% RSLogix 500 project slc_adjust_clock.RSS, saved by version 8.30.00.16 %
PROJECT "UNTITLED"    % processor: Bul.1763 MicroLogix 1100 Series B %

PROGRAM FILES
  LAD 2   4 rungs

DATA FILES
  O0 OUTPUT  4 elements
  I1 INPUT  6 elements
  S2 STATUS  66 elements
  B3 BINARY  1 elements
  T4 TIMER  1 elements
  C5 COUNTER  1 elements
  R6 CONTROL  1 elements
  N7 INTEGER  1 elements
  F8 FLOAT  1 elements
  N101 RTCBUFFERS  18 elements

LADDER 2
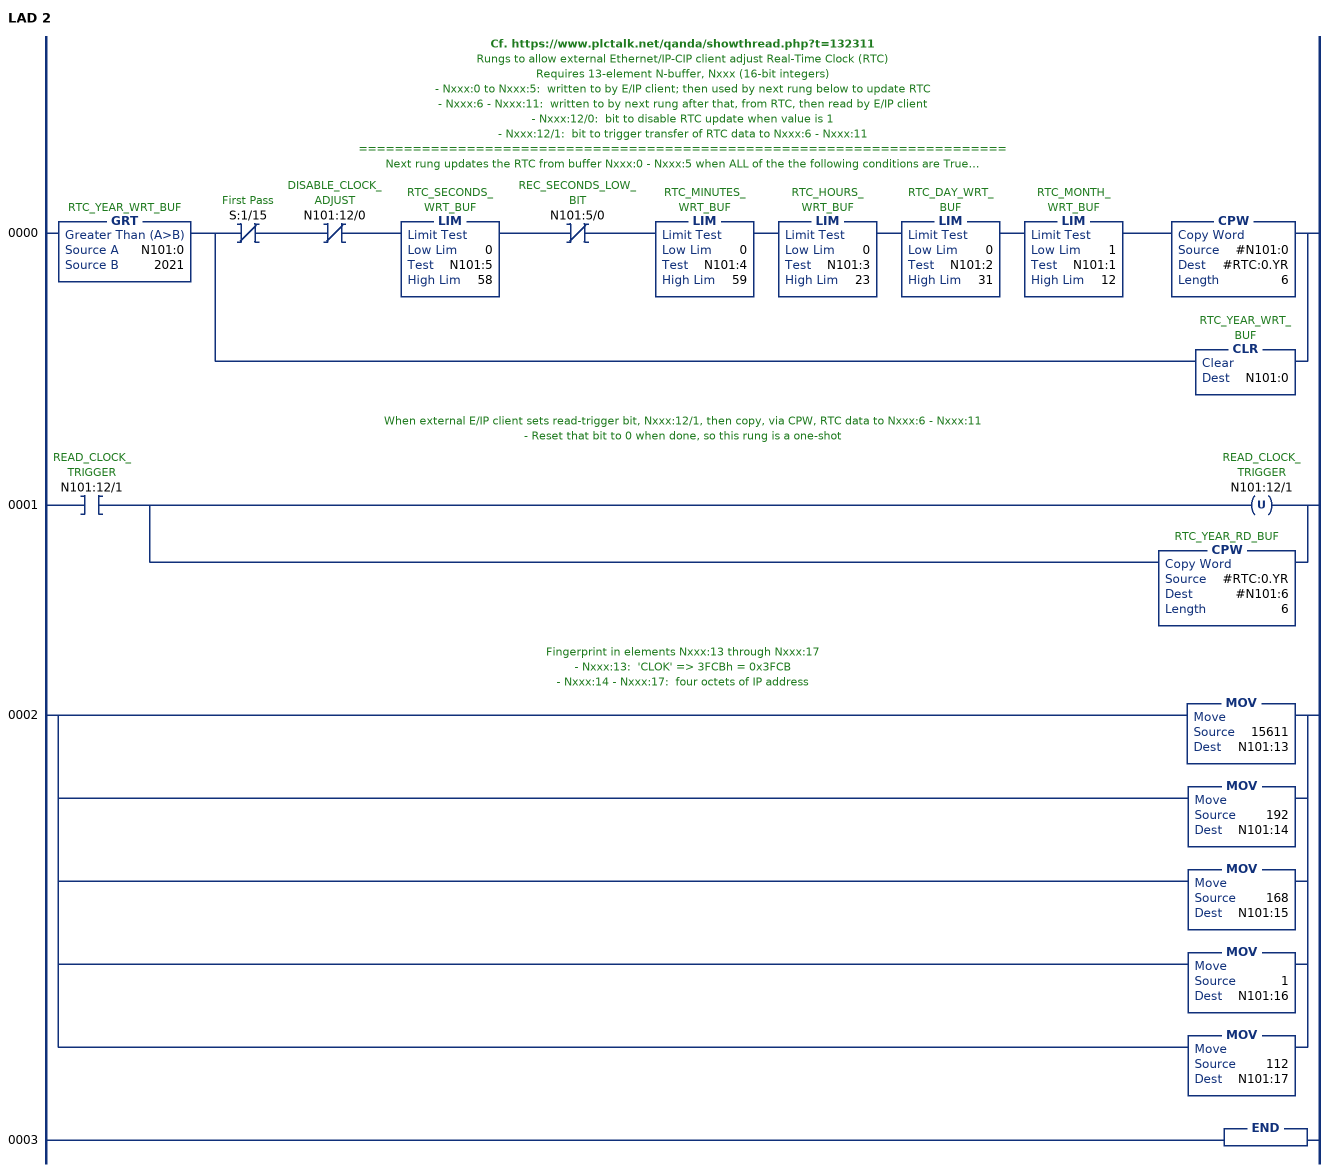
% Rung: 0 %
% TITLE: Cf. https://www.plctalk.net/qanda/showthread.php?t=132311 %
% Rungs to allow external Ethernet/IP-CIP client adjust Real-Time Clock (RTC)
% 
% Requires 13-element N-buffer, Nxxx (16-bit integers)
% - Nxxx:0 to Nxxx:5:  written to by E/IP client; then used by next rung below to update RTC
% - Nxxx:6 - Nxxx:11:  written to by next rung after that, from RTC, then read by E/IP client
% - Nxxx:12/0:  bit to disable RTC update when value is 1
% - Nxxx:12/1:  bit to trigger transfer of RTC data to Nxxx:6 - Nxxx:11
% 
% ========================================================================
% Next rung updates the RTC from buffer Nxxx:0 - Nxxx:5 when ALL of the the following conditions are True:
% - Buffered year is greater than 2021
% - This is not the First Pass scan
% - The clock adjustment is not disabled (Nxxx:12/0)
% - Buffered values are in valid ranges; also
%   - Value of seconds is even
%   - Value of day range is 1-31; no per-month or leap-year checks
% Next rung also assigns value of 0 to buffered year if it was greater than 2022,
% - this happens even if update to RTC does not execute, so this rung is a one-shot %
SOR GRT N101:0 2021 BST XIO S:1/15 XIO N101:12/0 LIM 0 N101:5 58 XIO N101:5/0 LIM 0 N101:4 59 LIM 0 N101:3 23 LIM 0 N101:2 31 LIM 1 N101:1 12 CPW #N101:0 #RTC:0.YR 6 NXB CLR N101:0 BND EOR
%   N101:0  RTC_YEAR_WRT_BUF %
%   S:1/15  "First Pass" %
%   N101:12/0  DISABLE_CLOCK_ADJUST %
%   N101:5  RTC_SECONDS_WRT_BUF %
%   N101:5/0  REC_SECONDS_LOW_BIT %
%   N101:4  RTC_MINUTES_WRT_BUF %
%   N101:3  RTC_HOURS_WRT_BUF %
%   N101:2  RTC_DAY_WRT_BUF %
%   N101:1  RTC_MONTH_WRT_BUF %
% Rung: 1 %
% When external E/IP client sets read-trigger bit, Nxxx:12/1, then copy, via CPW, RTC data to Nxxx:6 - Nxxx:11
% - Reset that bit to 0 when done, so this rung is a one-shot %
SOR XIC N101:12/1 BST OTU N101:12/1 NXB CPW #RTC:0.YR #N101:6 6 BND EOR
%   N101:12/1  READ_CLOCK_TRIGGER %
%   N101:6  RTC_YEAR_RD_BUF %
% Rung: 2 %
% Fingerprint in elements Nxxx:13 through Nxxx:17
% - Nxxx:13:  'CLOK' => 3FCBh = 0x3FCB
% - Nxxx:14 - Nxxx:17:  four octets of IP address %
SOR BST MOV 15611 N101:13 NXB MOV 192 N101:14 NXB MOV 168 N101:15 NXB MOV 1 N101:16 NXB MOV 112 N101:17 BND EOR
% Rung: 3 %
SOR END EOR

DATA TABLE (non-zero values as saved)
DATA T4
% .PRE .ACC %
% T4:0 % 3000 1246
DATA C5
% .PRE .ACC %
% C5:0 % 11 0
